Yaskawa INFORM job: A-4-08279-80-0-L.JBI

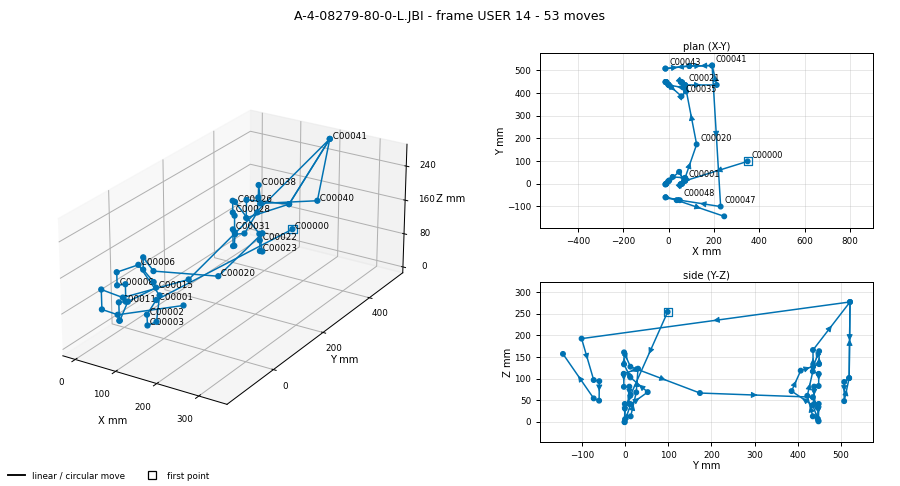
[picture p0: tool path of A-4-08279-80-0-L.JBI in frame USER 14, 53 of 53 moves have a stored position in this frame; points joined in program order, loops and branches not executed]
/JOB
//NAME A-4-08279-80-0-L
///FOLDERNAME PART_420-08279-80
//POS
///NPOS 53,0,53,0,0,0
///USER 14
///TOOL 4
///POSTYPE USER
///RECTAN
///RCONF 1,0,0,0,0,0,0,0,0,0,0,0,0,0,0,0,0,0,0,0,0,0,0,0
C00000=348.711,98.583,254.690,-96.7922,26.0608,130.3901
C00001=73.206,12.887,62.532,-108.1130,33.6440,124.7280
C00002=58.731,-0.654,30.802,-108.1124,33.6400,124.7315
C00003=59.251,-0.255,5.701,-108.1172,33.6444,124.7254
C00004=73.207,12.886,12.496,-108.1130,33.6440,124.7280
C00005=73.209,25.753,68.034,-108.1130,33.6440,124.7280
C00006=18.285,29.861,123.023,-105.1660,8.3780,132.7380
C00007=-13.751,-3.283,111.158,-105.6897,27.7501,134.0481
C00008=-13.813,-2.891,80.877,-102.0698,30.9749,134.6371
C00009=-1.744,9.833,81.413,-106.8820,26.9670,127.1640
C00010=-1.744,9.833,41.151,-106.8820,26.9670,127.1640
C00011=-12.048,-0.780,41.220,-105.8464,28.0451,133.0360
C00012=-11.621,-1.220,-1.083,-124.6790,17.6314,128.8686
C00013=-10.359,-1.214,-0.466,-124.6802,17.6302,128.8692
C00014=1.309,12.886,40.637,-115.9500,15.0640,123.8880
C00015=46.568,52.366,68.637,-115.9500,15.0640,123.8880
C00016=68.126,12.203,102.713,-51.9240,65.1860,170.4170
C00017=52.749,-2.584,132.935,-51.9209,65.1796,170.4256
C00018=53.344,-2.477,160.810,-51.9273,65.1792,170.4196
C00019=68.127,12.203,127.579,-51.9240,65.1860,170.4170
C00020=123.702,173.377,66.504,-51.9240,65.1860,170.4170
C00021=73.207,435.046,56.988,108.1130,33.6440,-124.7280
C00022=59.292,446.758,32.065,108.1131,33.6426,-124.7279
C00023=59.924,446.659,6.185,108.1129,33.6430,-124.7273
C00024=73.207,435.046,12.497,108.1130,33.6440,-124.7280
C00025=73.208,422.239,60.087,108.1130,33.6440,-124.7280
C00026=1.310,435.046,116.590,106.4700,24.0930,-128.1180
C00027=-13.463,448.705,111.098,105.5218,25.1062,-133.5890
C00028=-13.083,448.617,82.773,105.5202,25.1060,-133.5899
C00029=-1.744,438.100,81.414,106.4700,24.0930,-128.1180
C00030=-1.744,438.100,41.152,106.4700,24.0930,-128.1180
C00031=-13.002,448.729,41.356,105.1171,25.4810,-135.7662
C00032=-11.996,448.165,0.847,116.3410,16.2090,-135.3457
C00033=-8.859,448.159,2.300,116.3428,16.2080,-135.3458
C00034=1.310,435.046,37.856,114.8060,13.4990,-125.4170
C00035=56.824,385.802,71.014,114.8060,13.4990,-125.4170
C00036=76.829,406.941,118.422,51.9240,65.1860,-170.4170
C00037=53.293,449.586,133.474,51.9307,65.1846,-170.4129
C00038=53.934,449.681,163.520,51.9324,65.1847,-170.4119
C00039=68.127,435.729,127.579,51.9240,65.1860,-170.4170
C00040=212.373,435.445,166.233,51.9240,65.1860,-170.4170
C00041=191.994,521.318,277.669,-64.9580,52.3036,155.2869
C00042=91.520,519.266,101.171,-160.3299,74.1577,66.0982
C00043=-13.651,507.864,92.177,-160.3296,74.1566,66.1002
C00044=-14.273,507.713,47.691,-160.3275,74.1566,66.1021
C00045=91.520,519.266,101.171,-160.3299,74.1577,66.0982
C00046=191.994,521.318,277.669,-64.9580,52.3036,155.2869
C00047=229.653,-100.956,192.660,69.2460,43.0800,-149.5110
C00048=49.647,-72.877,96.659,69.2460,43.0800,-149.5110
C00049=-13.529,-59.896,94.020,69.2459,43.0778,-149.5114
C00050=-13.003,-60.326,48.795,69.2473,43.0797,-149.5114
C00051=35.736,-72.877,54.138,69.2460,43.0800,-149.5110
C00052=245.487,-144.122,157.206,69.2470,43.0790,-149.5110
///TOOL 0
///POSTYPE ANGLE
///ANGLE
EC00000=15.0000
///TOOL 4
EC00001=15.0000
///TOOL 0
EC00002=15.0000
EC00003=15.0000
///TOOL 4
EC00004=15.0000
EC00005=15.0000
EC00006=15.0000
///TOOL 0
EC00007=15.0000
EC00008=15.0000
///TOOL 4
EC00009=15.0000
EC00010=15.0000
///TOOL 0
EC00011=15.0000
EC00012=14.9994
EC00013=14.9994
///TOOL 4
EC00014=15.0000
EC00015=15.0000
EC00016=15.0000
///TOOL 0
EC00017=15.0000
EC00018=15.0000
///TOOL 4
EC00019=15.0000
EC00020=15.0000
EC00021=15.0000
///TOOL 0
EC00022=15.0000
EC00023=15.0000
///TOOL 4
EC00024=15.0000
EC00025=15.0000
EC00026=15.0000
///TOOL 0
EC00027=15.0000
EC00028=15.0000
///TOOL 4
EC00029=15.0000
EC00030=15.0000
///TOOL 0
EC00031=15.0000
EC00032=15.0000
EC00033=15.0000
///TOOL 4
EC00034=15.0000
EC00035=15.0000
EC00036=15.0000
///TOOL 0
EC00037=15.0000
EC00038=15.0000
///TOOL 4
EC00039=15.0000
EC00040=15.0000
///TOOL 0
EC00041=15.0000
EC00042=15.0000
EC00043=15.0000
EC00044=15.0000
EC00045=15.0000
EC00046=15.0000
///TOOL 4
EC00047=15.0000
EC00048=15.0000
///TOOL 0
EC00049=15.0000
EC00050=15.0000
///TOOL 4
EC00051=15.0000
EC00052=15.0000
//INST
///DATE 2021/10/29 11:36
///ATTR SC,RW,RJ
////FRAME USER 14
///GROUP1 RB1
///GROUP2 ST2
NOP
'Path Start: PP56
MOVJ C00000 VJ=100.00  +MOVJ EC00000
SMOVL C00001 V=1250.0  +MOVJ EC00001
SMOVL C00002 V=300.0  +MOVJ EC00002
ARCON ASF#(953)
SMOVL C00003 V=8.5  +MOVJ EC00003
ARCOF AEF#(953)
SMOVL C00004 V=1250.0  +MOVJ EC00004
SMOVL C00005 V=1250.0  +MOVJ EC00005
'Path End
'Path Start: PP54
SMOVL C00006 V=1250.0  +MOVJ EC00006
SMOVL C00007 V=300.0  +MOVJ EC00007
ARCON ASF#(952)
SMOVL C00008 V=6.3  +MOVJ EC00008
ARCOF AEF#(954)
SMOVL C00009 V=300.0  +MOVJ EC00009
SMOVL C00010 V=300.0  +MOVJ EC00010
SMOVL C00011 V=300.0  +MOVJ EC00011
ARCON ASF#(952)
SMOVL C00012 V=6.3  +MOVJ EC00012
SMOVL C00013 V=6.3  +MOVJ EC00013
ARCOF AEF#(952)
SMOVL C00014 V=1250.0  +MOVJ EC00014
SMOVL C00015 V=1250.0  +MOVJ EC00015
'Path End
'Path Start: Path_5
SMOVL C00016 V=1250.0  +MOVJ EC00016
SMOVL C00017 V=1250.0  +MOVJ EC00017
ARCON ASF#(951)
SMOVL C00018 V=8.5  +MOVJ EC00018
ARCOF AEF#(951)
SMOVL C00019 V=1250.0  +MOVJ EC00019
SMOVL C00020 V=1250.0  +MOVJ EC00020
'Path End
'Path Start: PP55
SMOVL C00021 V=1250.0  +MOVJ EC00021
SMOVL C00022 V=300.0  +MOVJ EC00022
ARCON ASF#(952)
SMOVL C00023 V=8.5  +MOVJ EC00023
ARCOF AEF#(952)
SMOVL C00024 V=1250.0  +MOVJ EC00024
SMOVL C00025 V=1250.0  +MOVJ EC00025
'Path End
'Path Start: PP58
SMOVL C00026 V=1250.0  +MOVJ EC00026
SMOVL C00027 V=300.0  +MOVJ EC00027
ARCON ASF#(952)
SMOVL C00028 V=6.3  +MOVJ EC00028
ARCOF AEF#(954)
SMOVL C00029 V=300.0  +MOVJ EC00029
SMOVL C00030 V=300.0  +MOVJ EC00030
SMOVL C00031 V=300.0  +MOVJ EC00031
ARCON ASF#(952)
SMOVL C00032 V=6.3  +MOVJ EC00032
SMOVL C00033 V=6.3  +MOVJ EC00033
ARCOF AEF#(952)
SMOVL C00034 V=1250.0  +MOVJ EC00034
SMOVL C00035 V=1250.0  +MOVJ EC00035
'Path End
'Path Start: Path_4
SMOVL C00036 V=1250.0  +MOVJ EC00036
SMOVL C00037 V=1250.0  +MOVJ EC00037
ARCON ASF#(951)
SMOVL C00038 V=8.5  +MOVJ EC00038
ARCOF AEF#(951)
SMOVL C00039 V=1250.0  +MOVJ EC00039
SMOVL C00040 V=1250.0  +MOVJ EC00040
'Path End
'Path Start: PP57
SMOVL C00041 V=1250.0  +MOVJ EC00041
SMOVL C00042 V=1250.0  +MOVJ EC00042
SMOVL C00043 V=300.0  +MOVJ EC00043
ARCON ASF#(953)
SMOVL C00044 V=10.6  +MOVJ EC00044
ARCOF AEF#(953)
SMOVL C00045 V=1250.0  +MOVJ EC00045
SMOVL C00046 V=1250.0  +MOVJ EC00046
'Path End
'Path Start: PP53
SMOVL C00047 V=1250.0  +MOVJ EC00047
SMOVL C00048 V=1250.0  +MOVJ EC00048
SMOVL C00049 V=300.0  +MOVJ EC00049
ARCON ASF#(953)
SMOVL C00050 V=10.6  +MOVJ EC00050
ARCOF AEF#(953)
SMOVL C00051 V=1250.0  +MOVJ EC00051
SMOVL C00052 V=1250.0  +MOVJ EC00052
'Path End
END
